Universal Robots PolyScope program: partmover02_subs.urp

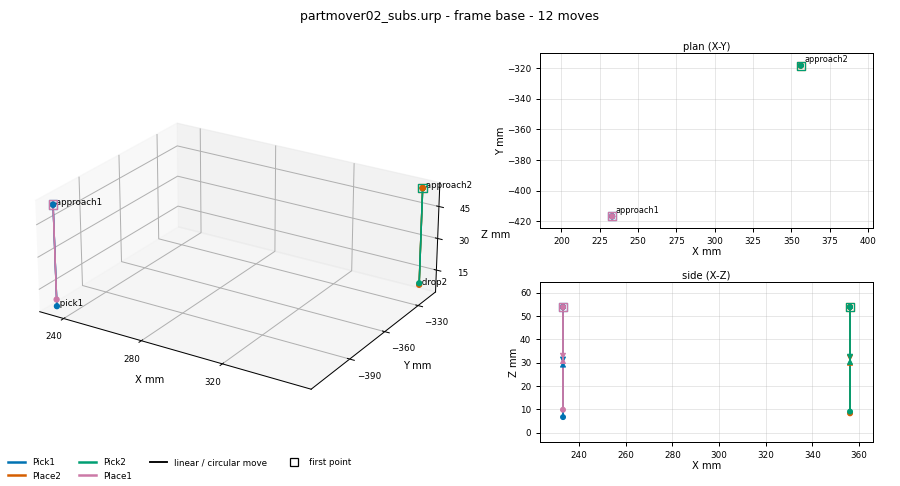
[picture p0: tool path of partmover02_subs.urp in frame base, 12 of 12 moves have a stored position in this frame; points joined in program order, loops and branches not executed]
Program partmover02_subs (installation=default directory=/programs createdIn=5.9.1.1031110 lastSavedIn=5.9.1.1031110 robotSerialNumber=20195501059)
Calibrated DH parameters: a=[0.000146, -0.418764, -0.053981, 0.000058, -0.000023, 0]; d=[0.162545, 37.319448, -206.067439, 168.881546, 0.09955, 0.099464]; alpha=[1.57004, -0.001979, 0.002304, 1.570607, -1.57066, 0]; deltaTheta=[0, -0.174616, -1.258233, 1.432844, -0.000001, 0]
BeforeStart
  URCap Gripper Activate (Robotiq_Grippers, Robotiq Inc.) dataModel(ResetAndActivateKey=false)
Robot Program (runOnlyOnce=true)
  Call Pick1
  Call Place2
  Call Pick2
  Call Place1
SubProgram -> Pick1
SubProgram -> Place2
SubProgram -> Pick2
SubProgram -> Place1
SubProgram Pick1 (keepSynchronizedWithDisk=false)
  MoveL speed 250 mm/s, acceleration 1200 mm/s^2 (useActiveTCP=true) feature=Base
    URCap Gripper (Robotiq_Grippers, Robotiq Inc.) dataModel(position=40.0, force=100.0, speed=100.0, positionInDouble=40.0, forceInDouble=100.0, speedInDouble=100.0, slaveIds=[9], blocking=false)
    Waypoint approach1: TCP in base x=233.098 y=-416.683 z=53.907 mm, rx=-2.1706 ry=-2.2616 rz=-0.0123 rad; joints [102.865, -81.519, 121.946, -129.844, 270.216, 100.549] deg; TCP offset x=0 y=0 z=174 mm, rx=0 ry=0 rz=0 rad
    Waypoint pick1: TCP in base x=233.126 y=-416.687 z=6.704 mm, rx=-2.1706 ry=-2.2616 rz=-0.0122 rad; joints [102.864, -76.18, 124.703, -137.941, 270.218, 100.559] deg
    URCap Gripper (Robotiq_Grippers, Robotiq Inc.) dataModel(position=100.0, force=100.0, speed=100.0, positionInDouble=100.0, forceInDouble=100.0, speedInDouble=100.0, slaveIds=[9], blocking=true)
    Waypoint approach1: TCP in base x=233.098 y=-416.683 z=53.907 mm, rx=-2.1706 ry=-2.2616 rz=-0.0123 rad; joints [102.865, -81.519, 121.946, -129.844, 270.216, 100.549] deg
SubProgram Place2 (keepSynchronizedWithDisk=false)
  MoveL speed 250 mm/s, acceleration 1200 mm/s^2 (useActiveTCP=true) feature=Base
    Waypoint approach2: TCP in base x=356.173 y=-318.335 z=53.911 mm, rx=-2.1706 ry=-2.2615 rz=-0.0123 rad; joints [121.755, -81.551, 122.012, -129.959, 270.395, 119.439] deg
    Waypoint drop2: TCP in base x=356.18 y=-318.346 z=8.327 mm, rx=-2.1707 ry=-2.2615 rz=-0.0123 rad; joints [121.75, -76.404, 124.688, -137.784, 270.397, 119.45] deg
    URCap Gripper (Robotiq_Grippers, Robotiq Inc.) dataModel(position=40.0, force=100.0, speed=100.0, positionInDouble=40.0, forceInDouble=100.0, speedInDouble=100.0, slaveIds=[9], blocking=true)
    Waypoint approach2: TCP in base x=356.173 y=-318.335 z=53.911 mm, rx=-2.1706 ry=-2.2615 rz=-0.0123 rad; joints [121.755, -81.551, 122.012, -129.959, 270.395, 119.439] deg
SubProgram Pick2 (keepSynchronizedWithDisk=false)
  MoveL speed 250 mm/s, acceleration 1200 mm/s^2 (useActiveTCP=true) feature=Base
    URCap Gripper (Robotiq_Grippers, Robotiq Inc.) dataModel(position=40.0, force=100.0, speed=100.0, positionInDouble=40.0, forceInDouble=100.0, speedInDouble=100.0, slaveIds=[9], blocking=false)
    Waypoint approach2: TCP in base x=356.173 y=-318.335 z=53.911 mm, rx=-2.1706 ry=-2.2615 rz=-0.0123 rad; joints [121.755, -81.551, 122.012, -129.959, 270.395, 119.439] deg
    Waypoint pick2: TCP in base x=356.182 y=-318.322 z=9.068 mm, rx=-2.1706 ry=-2.2616 rz=-0.0123 rad; joints [121.753, -76.495, 124.651, -137.653, 270.395, 119.449] deg
    URCap Gripper (Robotiq_Grippers, Robotiq Inc.) dataModel(position=100.0, force=100.0, speed=100.0, positionInDouble=100.0, forceInDouble=100.0, speedInDouble=100.0, slaveIds=[9], blocking=true)
    Waypoint approach2: TCP in base x=356.173 y=-318.335 z=53.911 mm, rx=-2.1706 ry=-2.2615 rz=-0.0123 rad; joints [121.755, -81.551, 122.012, -129.959, 270.395, 119.439] deg
SubProgram Place1 (keepSynchronizedWithDisk=false)
  MoveL speed 250 mm/s, acceleration 1200 mm/s^2 (useActiveTCP=true) feature=Base
    Waypoint approach1: TCP in base x=233.098 y=-416.683 z=53.907 mm, rx=-2.1706 ry=-2.2616 rz=-0.0123 rad; joints [102.865, -81.519, 121.946, -129.844, 270.216, 100.549] deg
    Waypoint drop1: TCP in base x=233.106 y=-416.692 z=9.863 mm, rx=-2.1706 ry=-2.2616 rz=-0.0122 rad; joints [102.863, -76.567, 124.546, -137.398, 270.215, 100.557] deg
    URCap Gripper (Robotiq_Grippers, Robotiq Inc.) dataModel(position=40.0, force=100.0, speed=100.0, positionInDouble=40.0, forceInDouble=100.0, speedInDouble=100.0, slaveIds=[9], blocking=true)
    Waypoint approach1: TCP in base x=233.098 y=-416.683 z=53.907 mm, rx=-2.1706 ry=-2.2616 rz=-0.0123 rad; joints [102.865, -81.519, 121.946, -129.844, 270.216, 100.549] deg
